INTERFACE I_DatatypeVisitor

METHOD VisitDatatype
VAR_INPUT
	VisitingDatatype : I_Datatype;
END_VAR
END_METHOD

END_INTERFACE

(* stored: Version 1.1.0.1, ProductVersion 3.1.4024.12
   Itf I_DatatypeVisitor: Id {75624d0e-5597-4f45-bcd9-af11f69a64ec}
   Method VisitDatatype: Id {77cdea5b-82f2-4c51-ba34-4afdde20d913} *)
